// TIA Portal V20 export
ORGANIZATION_BLOCK "Cyclic interrupt 1,5s"   // OB30, FBD, CyclicInterrupt
{ S7_Optimized_Access := 'TRUE' }
// stored: SetENOAutomatically false
   VAR_INPUT
      Initial_Call : Bool;   // Initial call of this OB
      Event_Count : Int;   // Events discarded
   END_VAR
BEGIN

NETWORK
TITLE = call diagnose
      CALL  "Diag", "Diag_DB";

END_ORGANIZATION_BLOCK
